// Mitsubishi GX Works2 project: 230928-002-COM UM BOTÃO   PLC: Q03UDV

// task Task_01 (event TRUE, interval 0, priority 31): POU_01

PROGRAM POU_01
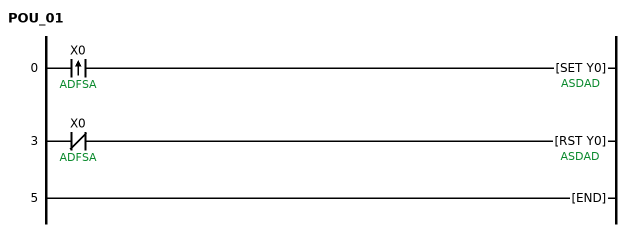
0     LDP     X0  ; ADFSA
      SET     Y0  ; ASDAD
3     LDI     X0  ; ADFSA
      RST     Y0  ; ASDAD
5     END
END_PROGRAM

// device comments not shown above
X1  ; ASDA
